TYPE ST_Event :
STRUCT
	eEventType : E_Type;
	eEventSeverity : TCEventSeverity;
	nEventDefinition : UINT;
	sEventMessage : STRING(255);
	tTimeStamp : DATE_AND_TIME;	
END_STRUCT
END_TYPE

(* stored: Version 1.1.0.1, ProductVersion 3.1.4024.9
   DUT ST_Event: Id {7e1c4e30-39f8-404e-b7cc-de3f99665e4d} *)
